{attribute addProperty BoxType "EPP1332-0001-0016"}
{attribute addProperty Id "A_0022_EPP1332_0001_0017A_0022_EPP1332_0001_0017_B713F54B2816352"}
{attribute addProperty CRC "218094176"}
{attribute addProperty SizeInBites "2816"}
{attribute addProperty SizeInBytes "352"}
TYPE A_0021_EPP1332_0001_0016_0CFFDA60 EXTENDS EPP1332_179A0949 :
STRUCT
	{attribute addProperty Name "A_0022_EPP1332_0001_0017"}
	A_0022_EPP1332_0001_0017 : A_0022_EPP1332_0001_0017_B713F54B;
END_STRUCT
END_TYPE

(* stored: Version 1.2.0.0, ProductVersion 3.1.4024.9
   DUT A_0021_EPP1332_0001_0016_0CFFDA60: Id {caf01197-b135-4896-b50b-6060fb5dbb74} *)
